{attribute 'GeneratedUsingTerminal: ELX4181-0000-0016'}
{attribute addProperty BoxType "ELX4181-0000-0016"}
{attribute addProperty Id "AO_OutputsAO_Outputs_BA7EBB7C2"}
{attribute addProperty CRC "2356519577"}
{attribute addProperty Size "2"}
TYPE Ch_1_8C75A299 :
STRUCT
	{attribute addProperty Name "AO_Outputs"}
	AO_Outputs  : AO_Outputs_BA7EBB7C;
END_STRUCT
END_TYPE

(* stored: Version 1.2.0.0, ProductVersion 3.1.4024.9
   DUT Ch_1_8C75A299: Id {13b68949-1bdb-4212-9e17-e177a24a9092} *)
